FUNCTION_BLOCK Grundablauf EXTENDS FB_Basis
VAR_INPUT
	// Instanzieren von Reaktor mit Interface
	Reaktor			:I_Reaktor;
	
	// Prozessparameter
	SekReaktor		:INT;
	Temp			:REAL;
	Entleermenge	:REAL;
	Pumpmenge		:REAL;
	Haltedauer		:TIME;
	Ruehrdauer		:TIME;
	Wartedauer		:TIME;
	Zirkulierdauer	:TIME;
END_VAR
VAR_OUTPUT
	
END_VAR
VAR
	LeitungsCheck	:BOOL := TRUE;
END_VAR

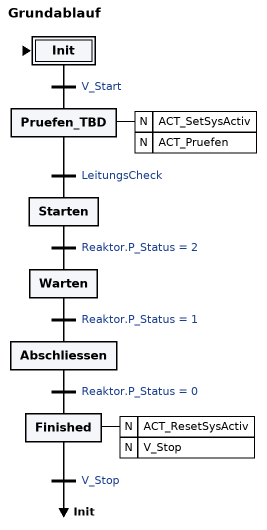
INITIAL_STEP Init:
END_STEP
TRANSITION FROM Init TO Pruefen_TBD
    := V_Start;
END_TRANSITION
STEP Pruefen_TBD:
    ACT_SetSysActiv(N);
    ACT_Pruefen(N);
END_STEP
TRANSITION FROM Pruefen_TBD TO Starten
    := LeitungsCheck;
END_TRANSITION
STEP Starten:
END_STEP
TRANSITION FROM Starten TO Warten
    := Reaktor.P_Status = 2;
END_TRANSITION
STEP Warten:
END_STEP
TRANSITION FROM Warten TO Abschliessen
    := Reaktor.P_Status = 1;
END_TRANSITION
STEP Abschliessen:
END_STEP
TRANSITION FROM Abschliessen TO Finished
    := Reaktor.P_Status = 0;
END_TRANSITION
STEP Finished:
    ACT_ResetSysActiv(N);
    V_Stop(N);
END_STEP
TRANSITION FROM Finished TO Init
    := V_Stop;
END_TRANSITION

ACTION ACT_Pruefen:
// TBD
END_ACTION

ACTION ACT_ResetSysActiv:
GVL.SysState := 0;
END_ACTION

ACTION ACT_SetSysActiv:
GVL.SysState := 1;
END_ACTION

END_FUNCTION_BLOCK

(* stored: Version 1.1.0.1, ProductVersion 3.1.4024.12
   POU Grundablauf: Id {ba376277-9321-4613-a760-dc59dad2be70}, SpecialFunc None
   Action ACT_Pruefen: Id {0cd24355-6c1e-4b69-9cae-0f7a68be8849}
   Action ACT_ResetSysActiv: Id {7cf457ea-1d08-461d-a894-7e22b2ced456}
   Action ACT_SetSysActiv: Id {efdd272f-178e-49f6-986a-deaf9af92096} *)
